// TIA Portal project "enkoder_lineer_sistem_kontrolu" (V18)

(* hardware
DEVICE "S7-1200 station_1"  S7-1200 Station
   slot 0: "Rack_0"  S7-1200 Rack  Rack  V1.0
   slot 1: "PLC_1"  CPU 1214C DC/DC/DC  6ES7 214-1AG40-0XB0  V4.6
*)

// ===== PLC "PLC_1"  CPU 1214C DC/DC/DC =====

VAR_GLOBAL   // PLC tag table "Default tag table"
   "Tag_1" AT %M20.0 : Bool;
   "Tag_2" AT %MD20 : DWord;
   "HSC5:P" AT %ID1016 : DWord;
   "HSC5 DEĞERİ" AT %MD2 : DWord;
   "START" AT %I0.0 : Bool;
   "START ÇIKIŞ" AT %Q0.0 : Bool;
   "VALVE" AT %Q1.0 : Bool;
   "ACİL ÇIKIŞ" AT %M70.0 : Bool;
   "HIZ" AT %I0.1 : Bool;
   "Tag_7" AT %Q0.3 : Bool;
   "YON" AT %Q0.1 : Bool;
   "Tag_3" AT %I0.7 : Bool;
END_VAR

// folder: System blocks/Program resources

DATA_BLOCK "T1"   // DB2
{ S7_Optimized_Access := 'TRUE' }
AUTHOR : Simatic
FAMILY : IEC
NAME : IEC_TMR
VERSION : 1.0
// stored: InstanceOfName IEC_TIMER
"IEC_TIMER"
BEGIN
END_DATA_BLOCK

// folder: (top level)

ORGANIZATION_BLOCK "Main"   // OB1, LAD, ProgramCycle
TITLE = "Main Program Sweep (Cycle)"
{ S7_Optimized_Access := 'TRUE' }
VERSION : 0.1
// A-B-Z fazli bir enkoder'in 1 turu 500 Pals'tir. Enkoder bir motorun miline baglidir. Motor Lineer bir sistemi hareket ettirmektedir. Motor, bir turnda lineer sistemi 0.1 cm hareket ettirmektedir. Lineer sistem 2 cm ileri hareket edecek ve duracaktir. Ayni anda çift etkili bir silindir, 5/2 tek tarafi selenoid valf ve geri dönüsümü yayl pnömatik bir valf araciligi ile hareket edecek, 3 saniye bekleyip geri hareket edecektir. Silindirin geri hareketi sonunda lineer sistem geri hareket edecek 0 cm yani baslangig noktasina geldiginde duracaktir.
// a. Gerekli hesaplamalari yapiniz.
// b. Proje tasarimini yapiniz.
// 
// 0.1 cm Lineer hareket için 500 pals gerekli
// 2cm lineer hareket için x pals gerekli
// 
// x=2*500/0.1= 10000 pulse gerekli
   VAR_INPUT
      Initial_Call : Bool;   // Initial call of this OB
      Remanence : Bool;   // =True, if remanent data are available
   END_VAR
   VAR_TEMP   // added for the SCL form of the ladder/FBD networks
      _w1 : Bool;
   END_VAR
BEGIN

REGION Network 1
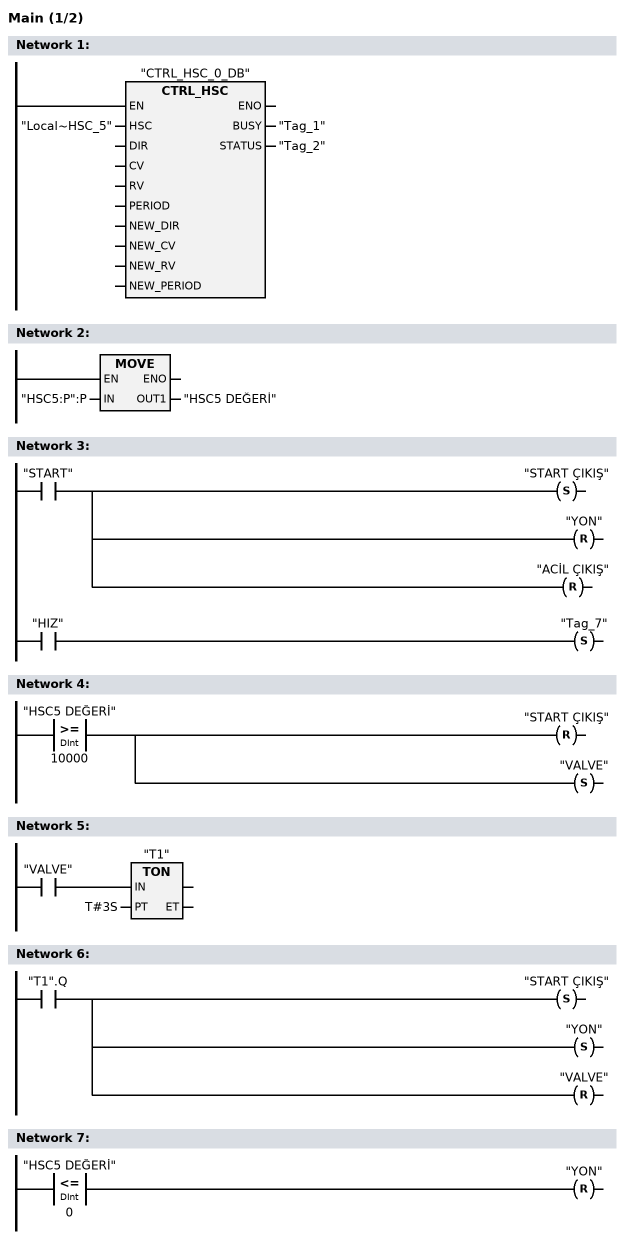
   "CTRL_HSC_0_DB"(HSC := "Local~HSC_5", BUSY => "Tag_1", STATUS => "Tag_2");   // CTRL_HSC
END_REGION

REGION Network 2
   RUNG wire#powerrail
      Move(in := "HSC5:P":P, out1 => "HSC5 DEĞERİ")
   END_RUNG
   // the same network as SCL:
   "HSC5 DEĞERİ" := "HSC5:P":P;
END_REGION

REGION Network 3
   RUNG wire#powerrail
      Contact( "START" )
      wire#w1
      S_Coil( "START ÇIKIŞ" )
   END_RUNG
   RUNG wire#w1
      R_Coil( "YON" )
   END_RUNG
   RUNG wire#w1
      R_Coil( "ACİL ÇIKIŞ" )
   END_RUNG
   RUNG wire#powerrail
      Contact( "HIZ" )
      S_Coil( "Tag_7" )
   END_RUNG
   // the same network as SCL:
   IF "START" THEN
       "START ÇIKIŞ" := TRUE;
       "YON" := FALSE;
       "ACİL ÇIKIŞ" := FALSE;
   END_IF;
   IF "HIZ" THEN "Tag_7" := TRUE; END_IF;
END_REGION

REGION Network 4
   RUNG wire#powerrail
      { S7_Templates := "SrcType := DInt" } GE_Contact(in1 := "HSC5 DEĞERİ", in2 := 10000)
      wire#w1
      R_Coil( "START ÇIKIŞ" )
   END_RUNG
   RUNG wire#w1
      S_Coil( "VALVE" )
   END_RUNG
   // the same network as SCL:
   IF "HSC5 DEĞERİ" >= 10000 THEN
       "START ÇIKIŞ" := FALSE;
       "VALVE" := TRUE;
   END_IF;
END_REGION

REGION Network 5
   "T1".TON(IN := "VALVE", PT := T#3S);
END_REGION

REGION Network 6
   RUNG wire#powerrail
      Contact( "T1".Q )
      wire#w1
      S_Coil( "START ÇIKIŞ" )
   END_RUNG
   RUNG wire#w1
      S_Coil( "YON" )
   END_RUNG
   RUNG wire#w1
      R_Coil( "VALVE" )
   END_RUNG
   // the same network as SCL:
   IF "T1".Q THEN
       "START ÇIKIŞ" := TRUE;
       "YON" := TRUE;
       "VALVE" := FALSE;
   END_IF;
END_REGION

REGION Network 7
   RUNG wire#powerrail
      { S7_Templates := "SrcType := DInt" } LE_Contact(in1 := "HSC5 DEĞERİ", in2 := 0)
      R_Coil( "YON" )
   END_RUNG
   // the same network as SCL:
   IF "HSC5 DEĞERİ" <= 0 THEN "YON" := FALSE; END_IF;
END_REGION

REGION Network 8
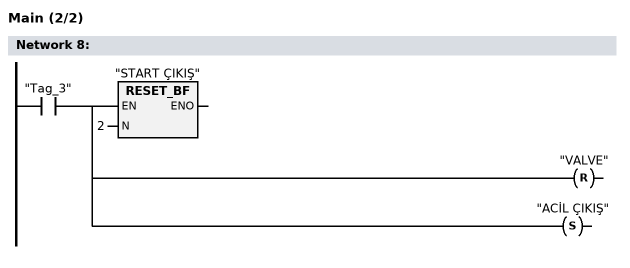
   // no SCL statement known for RBitfield: written as a call
   #_w1 := "Tag_3";
   IF #_w1 THEN
       RESET_BF(operand := "START ÇIKIŞ", n := 2);
       "VALVE" := FALSE;
       "ACİL ÇIKIŞ" := TRUE;
   END_IF;
END_REGION
END_ORGANIZATION_BLOCK